{attribute 'hide_all_locals'}
PROGRAM EthercatHelper
VAR
	fbReadDeviceName	: Tc2_IoFunctions.IOF_GetBoxNameByAddr;
	nMasterId			: UDINT;
END_VAR

// Converts Tc2_EtherCAT.ST_EcSlaveState to ZigaLibs_Core.ST_EcSlaveState and returns the converted structure.
METHOD ConvertBeckhoffEcStateToCustomStruct : ST_EcSlaveState
VAR_INPUT
	ecSlaveState	: Tc2_EtherCAT.ST_EcSlaveState;
END_VAR
VAR CONSTANT
	SLAVE_STATE_MASK 		: BYTE := 16#0F;
	SLAVE_STATE_EXTRAS_MASK : BYTE := 16#F0;
END_VAR
ConvertBeckhoffEcStateToCustomStruct.Device.State := SLAVE_STATE_MASK AND ecSlaveState.deviceState;
ConvertBeckhoffEcStateToCustomStruct.Device.StateExtras := SLAVE_STATE_EXTRAS_MASK AND ecSlaveState.deviceState;
ConvertBeckhoffEcStateToCustomStruct.Link := ecSlaveState.linkState;
END_METHOD

METHOD PUBLIC GetBoxNameByAddress : T_MaxString
VAR_INPUT
	PlcRuntimeNetId		: Tc2_System.T_AmsNetID; // NetId of the PLC where the devuce is located
	AmsNetId			: AMSADDR; // NetId of the box
	outError			: REFERENCE TO BOOL;	// If an error occurs while executing, method will provide the error flag here. This is a pointer to YOUR boolean error variable.
END_VAR

VAR
	sNetId	: Tc2_System.T_AmsNetID;
END_VAR
sNetId := AdsHelper.NetIdToString(AmsNetId.netId);
fbReadDeviceName(
	NETID := PlcRuntimeNetId,
	DEVICEID := AdsHelper.GetEthercatMasterIdFromNetIdString(netId := sNetId),
	BOXADDR := AmsNetId.port,
	START := NOT fbReadDeviceName.BUSY);
	
outError := fbReadDeviceName.ERR;
GetBoxNameByAddress := fbReadDeviceName.BOXNAME;
END_METHOD

END_PROGRAM

(* stored: Version 1.1.0.1, ProductVersion 3.1.4024.14
   POU EthercatHelper: Id {18c8e82e-8363-065e-3a67-80a80ad75944}, SpecialFunc None
   Method ConvertBeckhoffEcStateToCustomStruct: Id {902d4751-1f99-088d-257f-ddcd12172007}
   Method GetBoxNameByAddress: Id {05a15158-8102-075e-26df-9833faf2f947} *)
